TEXTLIST txtCylinderTypes
  0 = 'One Valve Spring Ret X2'
  1 = 'Two Valve Ret X3'
   = ''
END_TEXTLIST

(* stored: Version 1.1.0.1, ProductVersion 3.1.4019.2
   TextList txtCylinderTypes: Id {439625ab-bb57-4367-9ba1-6b0d9fedf0d0} *)
